KUKA KRL program: st1_st2.src

&ACCESS RVO1
&REL 4
&PARAM DISKPATH = KRC:\R1\Program\Moves\FROM_stPurge
DEF st1_st2 (lnPosNr :IN)
   DECL INT lnPosNr
   CONTINUE
   IF ($T1 OR $T2)THEN
      BAS(#INITMOV,0)
      PTP $POS_ACT
   ENDIF
   IF NOT (VARSTATE("lnPosNr") == #INITIALIZED) THEN
      lnPosNr = 1
   ENDIF

   xST1_ST2_10 = XST2
   eFromTmp = #ST1
   eToTmp = #ST2

   SWITCH lnPosNr
      CASE gnPosNr1
         GOTO Jump1
      CASE gnPosNr2
         GOTO Jump2
      CASE gnPosNr3
         GOTO Jump3
      CASE gnPosNr4
         GOTO Jump4
      CASE gnPosNr5
         GOTO Jump5
      CASE gnPosNr6
         GOTO Jump6
      CASE gnPosNr7
         GOTO Jump7
      CASE gnPosNr8
         GOTO Jump8
      CASE gnPosNr9
         GOTO Jump9
      CASE gnPosNr10
         GOTO Jump10
   ENDSWITCH

   Jump1:
   lnPosNr =gnPosNr1
   TRIGGER WHEN DISTANCE=0 DELAY=0 DO SaveLastPos(eFromTmp,eToTmp,gnPosNr1) PRIO=-1
   ;FOLD PTP xST1_ST2_1 CONT Vel= 100 % DATWork Tool[1] Base[0];%{PE}%R 5.4.35,%MKUKATPBASIS,%CMOVE,%VPTP,%P 1:PTP, 2:ST1_ST2_1, 3:C_PTP, 5:100, 7:DATWork
      $BWDSTART = FALSE
      PDAT_ACT=PDATWork
      FDAT_ACT=FST1_ST2_1
      BAS(#PTP_PARAMS,PDATWork.VEL)
      PTP xST1_ST2_1 C_PTP
   ;ENDFOLD

   Jump2:
   ;lnPosNr =gnPosNr2
   ;TRIGGER WHEN DISTANCE=0 DELAY=0 DO SaveLastPos(eFromTmp,eToTmp,gnPosNr2) PRIO=-1
   ;FOLD PTP xST1_ST2_2 CONT Vel= 100 % DATWork Tool[1] Base[0];%{PE}%R 5.4.35,%MKUKATPBASIS,%CMOVE,%VPTP,%P 1:PTP, 2:ST1_ST2_2, 3:C_PTP, 5:100, 7:DATWork
      ;$BWDSTART = FALSE
      ;PDAT_ACT=PDATWork
      ;FDAT_ACT=FST1_ST2_2
      ;BAS(#PTP_PARAMS,PDATWork.VEL)
      ;PTP xST1_ST2_2 C_PTP
   ;ENDFOLD

   Jump3:
   ;lnPosNr =gnPosNr3
   ;TRIGGER WHEN DISTANCE=0 DELAY=0 DO SaveLastPos(eFromTmp,eToTmp,gnPosNr3) PRIO=-1
   ;FOLD PTP xST1_ST2_3 CONT Vel= 100 % DATWork Tool[1] Base[0];%{PE}%R 5.4.35,%MKUKATPBASIS,%CMOVE,%VPTP,%P 1:PTP, 2:ST1_ST2_3, 3:C_PTP, 5:100, 7:DATWork
      ;$BWDSTART = FALSE
      ;PDAT_ACT=PDATWork
      ;FDAT_ACT=FST1_ST2_3
      ;BAS(#PTP_PARAMS,PDATWork.VEL)
      ;PTP xST1_ST2_3 C_PTP
   ;ENDFOLD

   Jump4:
   ;lnPosNr =gnPosNr4
   ;TRIGGER WHEN DISTANCE=0 DELAY=0 DO SaveLastPos(eFromTmp,eToTmp,gnPosNr4) PRIO=-1
   ;FOLD PTP xST1_ST2_4 CONT Vel= 100 % DATWork Tool[1] Base[0];%{PE}%R 5.4.35,%MKUKATPBASIS,%CMOVE,%VPTP,%P 1:PTP, 2:ST1_ST2_4, 3:C_PTP, 5:100, 7:DATWork
      ;$BWDSTART = FALSE
      ;PDAT_ACT=PDATWork
      ;FDAT_ACT=FST1_ST2_4
      ;BAS(#PTP_PARAMS,PDATWork.VEL)
      ;PTP xST1_ST2_4 C_PTP
   ;ENDFOLD

   Jump5:
   ;lnPosNr =gnPosNr5
   ;TRIGGER WHEN DISTANCE=0 DELAY=0 DO SaveLastPos(eFromTmp,eToTmp,gnPosNr5) PRIO=-1
   ;FOLD PTP xST1_ST2_5 CONT Vel= 100 % DATWork Tool[1] Base[0];%{PE}%R 5.4.35,%MKUKATPBASIS,%CMOVE,%VPTP,%P 1:PTP, 2:ST1_ST2_5, 3:C_PTP, 5:100, 7:DATWork
      ;$BWDSTART = FALSE
      ;PDAT_ACT=PDATWork
      ;FDAT_ACT=FST1_ST2_5
      ;BAS(#PTP_PARAMS,PDATWork.VEL)
      ;PTP xST1_ST2_5 C_PTP
   ;ENDFOLD

   Jump6:
   ;lnPosNr =gnPosNr6
   ;TRIGGER WHEN DISTANCE=0 DELAY=0 DO SaveLastPos(eFromTmp,eToTmp,gnPosNr6) PRIO=-1
   ;FOLD PTP xST1_ST2_6 CONT Vel= 100 % DATWork Tool[1] Base[0];%{PE}%R 5.4.35,%MKUKATPBASIS,%CMOVE,%VPTP,%P 1:PTP, 2:ST1_ST2_6, 3:C_PTP, 5:100, 7:DATWork
      ;$BWDSTART = FALSE
      ;PDAT_ACT=PDATWork
      ;FDAT_ACT=FST1_ST2_6
      ;BAS(#PTP_PARAMS,PDATWork.VEL)
      ;PTP xST1_ST2_6 C_PTP
   ;ENDFOLD

   Jump7:
   ;; lnPosNr =gnPosNr7
   ;; TRIGGER WHEN DISTANCE=0 DELAY=0 DO SaveLastPos(eFromTmp,eToTmp,gnPosNr7) PRIO=-1
   ;; ;FOLD PTP xST1_ST2_7 CONT Vel= 100 % DATWork Tool[1] Base[0];%{PE}%R 5.4.35,%MKUKATPBASIS,%CMOVE,%VPTP,%P 1:PTP, 2:ST1_ST2_7, 3:C_PTP, 5:100, 7:DATWork
   ;; $BWDSTART = FALSE
   ;; PDAT_ACT=PDATWork
   ;; FDAT_ACT=FST1_ST2_7
   ;; BAS(#PTP_PARAMS,PDATWork.VEL)
   ;; PTP xST1_ST2_7 C_PTP
   ;; ;ENDFOLD
   ;;
   Jump8:
   ;; lnPosNr =gnPosNr8
   ;; TRIGGER WHEN DISTANCE=0 DELAY=0 DO SaveLastPos(eFromTmp,eToTmp,gnPosNr8) PRIO=-1
   ;; ;FOLD PTP xST1_ST2_8 CONT Vel= 100 % DATWork Tool[1] Base[0];%{PE}%R 5.4.35,%MKUKATPBASIS,%CMOVE,%VPTP,%P 1:PTP, 2:ST1_ST2_8, 3:C_PTP, 5:100, 7:DATWork
   ;; $BWDSTART = FALSE
   ;; PDAT_ACT=PDATWork
   ;; FDAT_ACT=FST1_ST2_8
   ;; BAS(#PTP_PARAMS,PDATWork.VEL)
   ;; PTP xST1_ST2_8 C_PTP
   ;; ;ENDFOLD
   ;;
   Jump9:
   ;; lnPosNr =gnPosNr9
   ;; TRIGGER WHEN DISTANCE=0 DELAY=0 DO SaveLastPos(eFromTmp,eToTmp,gnPosNr9) PRIO=-1
   ;; ;FOLD PTP xST1_ST2_9 CONT Vel= 100 % DATWork Tool[1] Base[0];%{PE}%R 5.4.35,%MKUKATPBASIS,%CMOVE,%VPTP,%P 1:PTP, 2:ST1_ST2_9, 3:C_PTP, 5:100, 7:DATWork
   ;; $BWDSTART = FALSE
   ;; PDAT_ACT=PDATWork
   ;; FDAT_ACT=FST1_ST2_9
   ;; BAS(#PTP_PARAMS,PDATWork.VEL)
   ;; PTP xST1_ST2_9 C_PTP
   ;; ;ENDFOLD

   Jump10:
   lnPosNr =gnPosNr10
   TRIGGER WHEN DISTANCE=1 DELAY=0 DO SetStNumber() PRIO=-1
   TRIGGER WHEN DISTANCE=0 DELAY=0 DO SaveLastPos(eFromTmp,eToTmp,gnPosNr10) PRIO=-1
   ;FOLD PTP xST1_ST2_10 CONT Vel= 100 % DATWork Tool[1] Base[0];%{PE}%R 5.4.35,%MKUKATPBASIS,%CMOVE,%VPTP,%P 1:PTP, 2:ST1_ST2_10, 3:C_PTP, 5:100, 7:DATWork
      $BWDSTART = FALSE
      PDAT_ACT=PDATWork
      FDAT_ACT=FST1_ST2_10
      BAS(#PTP_PARAMS,PDATWork.VEL)
      PTP xST1_ST2_10 C_PTP
   ;ENDFOLD

END

DEF SetStNumber()
   gnActSt = 2
END
